KUKA KRL program: test.src, test.dat

--- test.src ---
&ACCESS RVP
&REL 90
&PARAM EDITMASK = *
&PARAM TEMPLATE = C:\KRC\Roboter\Template\vorgabe
&PARAM DISKPATH = KRC:\R1\Program
DEF test( )
;FOLD INI;%{PE}
  ;FOLD BASISTECH INI
    GLOBAL INTERRUPT DECL 3 WHEN $STOPMESS==TRUE DO IR_STOPM ( )
    INTERRUPT ON 3
    BAS (#INITMOV,0 )
  ;ENDFOLD (BASISTECH INI)
  ;FOLD USER INI
    ;Make your modifications here

  ;ENDFOLD (USER INI)
;ENDFOLD (INI)

;FOLD SPTP HOME CONT Vel=100 % DEFAULT ;%{PE}
;FOLD Parameters ;%{h}
;Params IlfProvider=kukaroboter.basistech.inlineforms.movement.spline; Kuka.IsGlobalPoint=False; Kuka.PointName=HOME; Kuka.BlendingEnabled=True; Kuka.MoveDataPtpName=DEFAULT; Kuka.VelocityPtp=100; Kuka.VelocityFieldEnabled=True; Kuka.ColDetectFieldEnabled=True; Kuka.CurrentCDSetIndex=0; Kuka.MovementParameterFieldEnabled=True; IlfCommand=SPTP
;ENDFOLD
SPTP XHOME WITH $VEL_AXIS[1] = SVEL_JOINT(100.0), $TOOL = STOOL2(FHOME), $BASE = SBASE(FHOME.BASE_NO), $IPO_MODE = SIPO_MODE(FHOME.IPO_FRAME), $LOAD = SLOAD(FHOME.TOOL_NO), $ACC_AXIS[1] = SACC_JOINT(PDEFAULT), $APO = SAPO_PTP(PDEFAULT), $GEAR_JERK[1] = SGEAR_JERK(PDEFAULT), $COLLMON_TOL_PRO[1] = USE_CM_PRO_VALUES(0) C_Spl
;ENDFOLD
REPEAT

ZATRZYMANIE_OPERATORSKIE()

;FOLD SPTP P1 Vel=100 % PDAT1 Tool[1]:TCP_WARSTWA Base[0] ;%{PE}
;FOLD Parameters ;%{h}
;Params IlfProvider=kukaroboter.basistech.inlineforms.movement.spline; Kuka.IsGlobalPoint=False; Kuka.PointName=P1; Kuka.BlendingEnabled=False; Kuka.MoveDataPtpName=PDAT1; Kuka.VelocityPtp=100; Kuka.VelocityFieldEnabled=True; Kuka.ColDetectFieldEnabled=True; Kuka.CurrentCDSetIndex=0; Kuka.MovementParameterFieldEnabled=True; IlfCommand=SPTP
;ENDFOLD
SPTP XP1 WITH $VEL_AXIS[1] = SVEL_JOINT(100.0), $TOOL = STOOL2(FP1), $BASE = SBASE(FP1.BASE_NO), $IPO_MODE = SIPO_MODE(FP1.IPO_FRAME), $LOAD = SLOAD(FP1.TOOL_NO), $ACC_AXIS[1] = SACC_JOINT(PPDAT1), $APO = SAPO_PTP(PPDAT1), $GEAR_JERK[1] = SGEAR_JERK(PPDAT1), $COLLMON_TOL_PRO[1] = USE_CM_PRO_VALUES(0)
;ENDFOLD

;PETLA OCZEKUJACA NA SYGNAL BEZ ZATRZYMANIA ROBOTA JEZELI WYSTAPI WCZESNIEJ
;$FLAG[1] = TRUE ; odczyt fiz wej zatrzymuje robota dlatego true
;IF ($FLAG[1] == FALSE) THEN
;  SPRAWDZ_IN(1)
;ENDIF
REPEAT
UNTIL($FLAG[1])

ZAJECIE_STR_KOL(2,2)
ZAJECIE_STR_PLC(3,4)

;FOLD SPTP P2 CONT Vel=100 % PDAT2 Tool[1]:TCP_WARSTWA Base[0] ;%{PE}
;FOLD Parameters ;%{h}
;Params IlfProvider=kukaroboter.basistech.inlineforms.movement.spline; Kuka.IsGlobalPoint=False; Kuka.PointName=P2; Kuka.BlendingEnabled=True; Kuka.MoveDataPtpName=PDAT2; Kuka.VelocityPtp=100; Kuka.VelocityFieldEnabled=True; Kuka.ColDetectFieldEnabled=True; Kuka.CurrentCDSetIndex=0; Kuka.MovementParameterFieldEnabled=True; IlfCommand=SPTP
;ENDFOLD
SPTP XP2 WITH $VEL_AXIS[1] = SVEL_JOINT(100.0), $TOOL = STOOL2(FP2), $BASE = SBASE(FP2.BASE_NO), $IPO_MODE = SIPO_MODE(FP2.IPO_FRAME), $LOAD = SLOAD(FP2.TOOL_NO), $ACC_AXIS[1] = SACC_JOINT(PPDAT2), $APO = SAPO_PTP(PPDAT2), $GEAR_JERK[1] = SGEAR_JERK(PPDAT2), $COLLMON_TOL_PRO[1] = USE_CM_PRO_VALUES(0) C_Spl
;ENDFOLD

;FOLD SPTP HOME Vel=100 % DEFAULT ;%{PE}
;FOLD Parameters ;%{h}
;Params IlfProvider=kukaroboter.basistech.inlineforms.movement.spline; Kuka.IsGlobalPoint=False; Kuka.PointName=HOME; Kuka.BlendingEnabled=False; Kuka.MoveDataPtpName=DEFAULT; Kuka.VelocityPtp=100; Kuka.VelocityFieldEnabled=True; Kuka.ColDetectFieldEnabled=True; Kuka.CurrentCDSetIndex=0; Kuka.MovementParameterFieldEnabled=True; IlfCommand=SPTP
;ENDFOLD
SPTP XHOME WITH $VEL_AXIS[1] = SVEL_JOINT(100.0), $TOOL = STOOL2(FHOME), $BASE = SBASE(FHOME.BASE_NO), $IPO_MODE = SIPO_MODE(FHOME.IPO_FRAME), $LOAD = SLOAD(FHOME.TOOL_NO), $ACC_AXIS[1] = SACC_JOINT(PDEFAULT), $APO = SAPO_PTP(PDEFAULT), $GEAR_JERK[1] = SGEAR_JERK(PDEFAULT), $COLLMON_TOL_PRO[1] = USE_CM_PRO_VALUES(0)
;ENDFOLD

UNTIL ($FLAG[2])
END

DEF ZAJECIE_STR_KOL(NR_WYJ:IN,NR_WEJ:IN)

DECL INT NR_WYJ
DECL INT NR_WEJ

  ;REQUEST
  $OUT[NR_WYJ]=TRUE
  ;TAKE WORK AREA
  WAIT FOR $IN[NR_WEJ]

END

DEF ZAJECIE_STR_PLC(NR_WYJ:IN, NR_WEJ:IN)

DECL INT NR_WYJ
DECL INT NR_WEJ

  ;REQUEST
  $OUT[NR_WYJ]=TRUE
  ;TAKE COLISION ZONE
  WAIT FOR $IN[NR_WEJ]

END

DEF ZATRZYMANIE_OPERATORSKIE()

  IF($IN[100]) THEN
    $OUT[100]=TRUE
    WAIT FOR (NOT $IN[100])
    $OUT[100]=FALSE
  ENDIF

END

DEF SPRAWDZ_IN(NR_WEJ:IN)
DECL INT NR_WEJ

REPEAT

UNTIL($IN[NR_WEJ])

END

--- test.dat ---
&ACCESS RVP
&REL 90
&PARAM EDITMASK = *
&PARAM TEMPLATE = C:\KRC\Roboter\Template\vorgabe
&PARAM DISKPATH = KRC:\R1\Program
DEFDAT  TEST
;FOLD EXTERNAL DECLARATIONS;%{PE}%MKUKATPBASIS,%CEXT,%VCOMMON,%P
;FOLD BASISTECH EXT;%{PE}%MKUKATPBASIS,%CEXT,%VEXT,%P
EXT  BAS (BAS_COMMAND  :IN,REAL  :IN )
DECL INT SUCCESS
;ENDFOLD (BASISTECH EXT)
;FOLD USER EXT;%{E}%MKUKATPUSER,%CEXT,%VEXT,%P
;Make your modifications here

;ENDFOLD (USER EXT)
;ENDFOLD (EXTERNAL DECLARATIONS)
DECL E6POS XP1={X 1362.21301,Y -2097.62402,Z 642.604614,A -147.000,B 2.29571695E-09,C -167.192444,S 2,T 10,E1 0.0,E2 0.0,E3 0.0,E4 0.0,E5 0.0,E6 0.0}
DECL FDAT FP1={TOOL_NO 1,BASE_NO 0,IPO_FRAME #BASE,POINT2[] " "}
DECL PDAT PPDAT1={VEL 100.000,ACC 100.000,APO_DIST 500.000,APO_MODE #CDIS,GEAR_JERK 100.000,EXAX_IGN 0}
DECL MODULEPARAM_T LAST_TP_PARAMS={PARAMS[] "Kuka.VelocityFieldEnabled=True; Kuka.ColDetectFieldEnabled=True; Kuka.MovementParameterFieldEnabled=True; Kuka.IsAngleEnabled=False; Kuka.PointName=P1; Kuka.FrameData.base_no=0; Kuka.FrameData.tool_no=1; Kuka.FrameData.ipo_frame=#BASE; Kuka.isglobalpoint=False; Kuka.MoveDataPtpName=PDAT1; Kuka.MovementDataPdat.apo_mode=#CDIS; Kuka.MovementDataPdat.apo_dist=500; Kuka.MovementData.vel=100; Kuka.MovementData.acc=100; Kuka.MovementData.gear_jerk=100; Kuka.MovementData.exax_ign=0; Kuka.VelocityPtp=100; Kuka.BlendingEnabled=False; Kuka.CurrentCDSetIndex=0; Kuka.FrameData.point2=     "}
DECL E6POS XP2={X 1012.38586,Y -2287.07813,Z 642.604614,A -156.123199,B 3.98594491E-09,C -167.192444,S 2,T 10,E1 0.0,E2 0.0,E3 0.0,E4 0.0,E5 0.0,E6 0.0}
DECL FDAT FP2={TOOL_NO 1,BASE_NO 0,IPO_FRAME #BASE,POINT2[] " "}
DECL PDAT PPDAT2={VEL 100.000,ACC 100.000,APO_DIST 500.000,APO_MODE #CDIS,GEAR_JERK 100.000,EXAX_IGN 0}
ENDDAT
